// TIA Portal V17 export
// export: Created 2024-08-07T21:44:14.0379756Z, ExportSetting WithDefaults, DisplayName Totally Integrated Automation Portal, DisplayVersion V17 Update 7, DisplayName TIA Portal Openness, DisplayVersion V17 Update 7, DisplayName TIA Portal Version Control Interface, DisplayVersion V17, DisplayName SINAMICS Startdrive Advanced, DisplayVersion V17 SP2, DisplayName SINAMICS Startdrive G110M, G120, G120C, G120D, G120P, G115D, DisplayVersion V17 SP2, DisplayName SINAMICS Startdrive G130, G150, S120, S150, SINAMICS MV, S210, DisplayVersion V17 SP2, DisplayName STEP 7 Professional, DisplayVersion V17 Update 7, DisplayName STEP 7 Safety, DisplayVersion V17 Update 6, DisplayName WinCC Advanced / Unified PC, DisplayVersion V17 Update 7
TYPE "UDT_PositionData"
// stored: IsFailsafeCompliant false
   STRUCT
      PartPresent : Bool;
      PartNOK : Bool;
      PartErrors : Array[0..255] of Bool;
      Reference : Int;
      FinishedOperations : Array[0..15] of Bool;
      StFinished : Array[0..15] of Bool;
      Scan : String[30];
      IJCType : Int;   // 0 - no ijc; 1 - Standart IJC; 2 - P variant; 3 - downgrade mode
      CreatedNFP : Array[1.."MaxCreateNFP"] of String[30];
      Readings : Array[1.."MaxDataReading"] of Struct
         Scan : String[70];
      END_STRUCT;
   END_STRUCT;
END_TYPE
